// TIA Portal V17 export
// export: Created 2024-10-17T14:16:18.3201486Z, ExportSetting WithDefaults, DisplayName Totally Integrated Automation Portal, DisplayVersion V17 Update 4, DisplayName TIA Portal Openness, DisplayVersion V17 Update 4, DisplayName TIA Portal Version Control Interface, DisplayVersion V17, DisplayName SINAMICS Startdrive Advanced, DisplayVersion V17 Update2, DisplayName SINAMICS Startdrive G130, G150, S120, S150, SINAMICS MV, S210, DisplayVersion V17 Update2, DisplayName SINAMICS Startdrive G110M, G120, G120C, G120D, G120P, G115D, DisplayVersion V17 Update2, DisplayName STEP 7 Professional, DisplayVersion V17 Update 4, DisplayName STEP 7 Safety, DisplayVersion V17, DisplayName WinCC Advanced / Unified PC, DisplayVersion V17 Update 4
TYPE "LPMLV2022_typeParameter_STRING"
TITLE = LPMLV2022_typeParameter_STRING
// Support: tech.team.motioncontrol@siemens.com
// stored: IsFailsafeCompliant false
   STRUCT
      ID : DInt;   // ID Value of Parameter. This is the arbitrary (user defined) ID value of the parameter
      "Name" : String[80];   // Name of Parameter. The literal parameter name is used to describe the parameter number, and its associated value
      Unit : String[6];   // Unit of Measure of Parameter. The parameter unit is typically not used for string values
      Value : String[80];   // Value of Parameter. This is the string value of the parameter
   END_STRUCT;
END_TYPE
